// TIA Portal V20 export
VAR_GLOBAL   // PLC tag table "Default tag table"
   "Pump running" AT %Q0.1 : Bool;
END_VAR
VAR_GLOBAL CONSTANT   // user constants
   C_MAX : Int := 4;
END_VAR
